(* IEC 61131-3 sources: statemachine/src/StateFramework/Guards, 10 files *)

(* ---- CompareGuardLint.st ---- *)
NAMESPACE Simatic.Ax.StateFramework

    /// Condition
    /// GT: Greater than compareValue
    /// EQ: Equal to compareValue
    /// LT: Less than compareValue
    /// NE: Is not equal to compareValue
    /// GE: Greater or equal to compareValue
    /// LE: Less or equal to compareValue
    TYPE
        Condition : (GT, EQ, LT, NE, GE, LE);
    END_TYPE

    CLASS CompareGuardLint IMPLEMENTS IGuard
        VAR PUBLIC
            // Referenced runtime value that is compared against CompareToValue.
            Value : REF_TO LINT;
            // Constant comparison target.
            CompareToValue : LINT;
            // Selected comparison operator.
            Condition : Condition;
        END_VAR

        METHOD PUBLIC Config
            VAR_INPUT
                countValue : REF_TO LINT;
                compareValue : LINT;
                compareCondition : Condition;
            END_VAR
            // Config stores the referenced value, threshold and comparison mode.
            Value := countValue;
            CompareToValue := compareValue;
            Condition := compareCondition;
        END_METHOD

        METHOD PUBLIC Check : BOOL
            // The referenced value is evaluated with the configured comparison operator.
            CASE Condition OF
                Condition#GT : Check := Value^ > CompareToValue;
                Condition#EQ : Check := Value^ = CompareToValue;
                Condition#LT : Check := Value^ < CompareToValue;
                Condition#GE : Check := Value^ >= CompareToValue;
                Condition#LE : Check := Value^ <= CompareToValue;
            END_CASE
            ;

        END_METHOD

        METHOD PUBLIC Reset
            // CompareGuardLint is stateless and therefore does not need a reset action.
            ;
        END_METHOD

    END_CLASS
END_NAMESPACE

(* ---- IGuard.st ---- *)
NAMESPACE Simatic.Ax.StateFramework
    INTERFACE IGuard

        // Evaluates the guard condition for the current cycle.
        METHOD Check : BOOL
        END_METHOD

        // Resets any internal state kept by the guard.
        METHOD Reset
        END_METHOD

    END_INTERFACE
END_NAMESPACE

(* ---- AndGuard.st ---- *)
NAMESPACE Simatic.Ax.StateFramework
    /// AND Guard
    ///   Lhs : IGuard;
    ///   Rhs : IGuard;
    /// Rhs and Lhs must be TRUE that the Check()-Method returns true
    {axcode:docs-v0:@simatic-ax/statemachine:AndGuard.md}
    CLASS AndGuard IMPLEMENTS IGuard
        VAR PUBLIC
            Lhs : IGuard;
            Rhs : IGuard;
        END_VAR

        METHOD PUBLIC Check : BOOL
            IF (Lhs = NULL) OR (Rhs = NULL) THEN
                Check := FALSE;
            ELSE
                Check := Lhs.Check() AND Rhs.Check();
            END_IF;
        END_METHOD

        METHOD PUBLIC Reset
            IF (Lhs <> NULL) THEN
                Lhs.Reset();
            END_IF;
            IF (Rhs <> NULL) THEN
                Rhs.Reset();
            END_IF;
        END_METHOD

    END_CLASS
END_NAMESPACE

(* ---- BoolGuard.st ---- *)
NAMESPACE Simatic.Ax.StateFramework
    /// BOOL Guard
    /// Value : REF_TO BOOL
    /// Check()-Method returns true when REF_TO value is TRUE
    CLASS BoolGuard IMPLEMENTS IGuard
        VAR PUBLIC
            Value : REF_TO BOOL;
        END_VAR

        METHOD PUBLIC Check : BOOL
            IF (Value = NULL) THEN
                Check := FALSE;
            ELSE
                Check := Value^;
            END_IF;
        END_METHOD

        METHOD PUBLIC Reset
            ;
        END_METHOD

    END_CLASS
END_NAMESPACE

(* ---- CountGuard.st ---- *)
NAMESPACE Simatic.Ax.StateFramework

    CLASS CountGuard IMPLEMENTS IGuard
        VAR PUBLIC
            Count : LINT;
        END_VAR
        VAR
            _actCount : LINT;
        END_VAR

        METHOD PUBLIC Config
            VAR_INPUT
                countValue : LINT;
            END_VAR
            // Count defines after how many Check calls the guard becomes TRUE once.
            Count := countValue;
        END_METHOD

        METHOD PUBLIC Check : BOOL
            // The counter is incremented on every evaluation and resets after firing.
            _actCount := _actCount + LINT#1;
            IF (_actCount >= Count) THEN
                _actCount := LINT#0;
                Check := TRUE;
            ELSE
                Check := FALSE;
            END_IF;

        END_METHOD

        METHOD PUBLIC Reset
            // CountGuard keeps counting across cycles until it fires.
            ;
        END_METHOD

    END_CLASS

END_NAMESPACE

(* ---- NotGuard.st ---- *)
NAMESPACE Simatic.Ax.StateFramework
    CLASS NotGuard IMPLEMENTS IGuard
        VAR PUBLIC
            Guard : IGuard;
        END_VAR

        METHOD PUBLIC Check : BOOL
            IF (Guard = NULL) THEN
                Check := FALSE;
            ELSE
                Check := NOT(Guard.Check());
            END_IF;
        END_METHOD

        METHOD PUBLIC Reset
            IF (Guard <> NULL) THEN
                Guard.Reset();
            END_IF;
        END_METHOD

    END_CLASS
END_NAMESPACE

(* ---- OrGuard.st ---- *)
NAMESPACE Simatic.Ax.StateFramework
    CLASS OrGuard IMPLEMENTS IGuard
        VAR PUBLIC
            Lhs : IGuard;
            Rhs : IGuard;
        END_VAR

        METHOD PUBLIC Check : BOOL
            IF (Lhs = NULL) AND (Rhs = NULL) THEN
                Check := FALSE;
            ELSIF (Lhs = NULL) THEN
                Check := Rhs.Check();
            ELSIF (Rhs = NULL) THEN
                Check := Lhs.Check();
            ELSE
                Check := Lhs.Check() OR Rhs.Check();
            END_IF;
        END_METHOD

        METHOD PUBLIC Reset
            IF (Lhs <> NULL) THEN
                Lhs.Reset();
            END_IF;
            IF (Rhs <> NULL) THEN
                Rhs.Reset();
            END_IF;
        END_METHOD

    END_CLASS
END_NAMESPACE

(* ---- TimeoutGuard.st ---- *)
USING System.Timer;

NAMESPACE Simatic.Ax.StateFramework

    CLASS TimeoutGuard IMPLEMENTS IGuard
        VAR PUBLIC
            Timeout : TIME;
        END_VAR
        VAR
            _ton : OnDelay;
        END_VAR

        METHOD PUBLIC Config
            VAR_INPUT
                timeoutValue : TIME;
            END_VAR
            // Timeout defines the TON duration that must elapse before Check returns TRUE.
            Timeout := timeoutValue;
        END_METHOD

        METHOD PUBLIC Check : BOOL
            // The timer is driven continuously until the configured delay has elapsed.
            _ton(signal := TRUE, duration := Timeout);
            IF (_ton.output) THEN
                 Check := TRUE;
            ELSE
                Check := FALSE;
            END_IF;
        END_METHOD

        METHOD PUBLIC Reset
            // Reset drops the TON input so the timeout starts from zero on the next Check.
            _ton(signal:= FALSE);
        END_METHOD

    END_CLASS
END_NAMESPACE

(* ---- TrueGuard.st ---- *)
NAMESPACE Simatic.Ax.StateFramework

    CLASS TrueGuard IMPLEMENTS IGuard
        METHOD PUBLIC Check : BOOL
            // This guard is always open.
            Check := TRUE;
        END_METHOD

        METHOD PUBLIC Reset
            // TrueGuard has no internal state to reset.
            ;
        END_METHOD

    END_CLASS
END_NAMESPACE

(* ---- XorGuard.st ---- *)
NAMESPACE Simatic.Ax.StateFramework
    CLASS XorGuard IMPLEMENTS IGuard
        VAR PUBLIC
            Lhs : IGuard;
            Rhs : IGuard;
        END_VAR

        METHOD PUBLIC Check : BOOL
            IF (Lhs = NULL) AND (Rhs = NULL) THEN
                Check := FALSE;
            ELSIF (Lhs = NULL) THEN
                Check := Rhs.Check();
            ELSIF (Rhs = NULL) THEN
                Check := Lhs.Check();
            ELSE
                Check := Lhs.Check() XOR Rhs.Check();
            END_IF;
        END_METHOD

        METHOD PUBLIC Reset
            IF (Lhs <> NULL) THEN
                Lhs.Reset();
            END_IF;
            IF (Rhs <> NULL) THEN
                Rhs.Reset();
            END_IF;
        END_METHOD

    END_CLASS
END_NAMESPACE
